INTERFACE I_GraphVisitor

METHOD VisitGraph
VAR_INPUT
	VisitingGraph : I_Graph;
END_VAR
END_METHOD

END_INTERFACE

(* stored: Version 1.1.0.1, ProductVersion 3.1.4024.12
   Itf I_GraphVisitor: Id {8f09db5b-eb4f-46b4-8dcb-6f37fa95677f}
   Method VisitGraph: Id {45f8c81d-001c-429e-bb38-1b3935bcfeee} *)
